(* IEC 61131-3 sources: CodigoPPC/FB Controle, 12 files *)

(* ---- FB_Controle.st ---- *)
(*
   FB_Controle: Bloco Principal de Controle de Exportação (Zero Grid / Limitação).

   OBJETIVO:
   Gerenciar a potência ativa e reativa dos inversores para garantir que a exportação
   de energia no ponto de conexão (PCC) não ultrapasse os limites definidos na agenda.

   ESTRATÉGIA DE CONTROLE (Lógica Inversa):
   - PV (Process Variable) é o valor medido no ponto de conexão
     - Valor Positivo (+) = Importando da rede (Consumo > Geração).
     - Valor Negativo (-) = Exportando para rede (Geração > Consumo).
   - SP (Set Point) é o limite de exportação (ex: -50kW).
   - O PID atua para manter PV >= SP.
     - Se PV > SP (Importando), o PID aumenta a geração.
     - Se PV < SP (Exportando), o PID reduz a geração.
	 Controle de Exportação em kW (Zero = Autoconsumo, Negativo = Exportação, Positivo = Importação).
	Erro: SP - PV.
	Ex: Quero exportar -10kW. Medidor lê +5kW (Importando). Erro = -10 - 5 = -15.
	Para aumentar a geração (reduzir a importação), o PID precisa agir.
	Atenção: Como o comando do inversor é sempre positivo (0..100% de geração), a lógica interna do PI deve ser Inversa (Erro negativo -> Aumenta Saída) ou ajustamos o sinal do erro na entrada.

	No código abaixo, a estratégia usada foi de Normalizar o Erro para "Quanto falta gerar".
	Se o medidor diz +10kW (Importando), precisamos gerar +10kW a mais.
	Se o medidor diz -20kW (Exportando muito) e o limite é -10kW, precisamos gerar 10kW a menos.

    Hierarquia de prioridades ou objetivos:

    Prioridade 1: MAXIMIZAR P (Potência Ativa)
	Objetivo: Gerar o máximo de potência ativa possível
	Limite: Exportação máxima (agenda + safety margin + limite de fase)
	Flexibilidade: RÍGIDO - nunca exceder

	Prioridade 2: PF ≥ 0.92 NO PONTO DE CONEXÃO
	Objetivo: Manter fator de potência ≥ 0.92 (indutivo)
	Método: Compensar Q da carga com Q dos inversores
	Flexibilidade: SOFT - sinaliza se não conseguir, mas NÃO reduz P

	Prioridade 3: BALANCEAMENTO DE FASES

    Ordem de execução:
	0. Leitura do medidor e ajuste dos valores para unidades corretas
	Lê registradores Modbus, converte e armazena como variáveis Globais

	Dentro de FB_Controle
	1. FB_Scheduler - Define limite de exportação baseado em datas, dias de semana e horário
    2. FB_PowertController
		2.1. PI → P_cmd_raw
    	2.2. Safety Margin → P_cmd_with_margin
    	2.3. Limitador de Fase → P_cmd_limited
    3. FB_FFQ - Feedforward de Q (estimativa inicial)
    4. FB_PIQ - Controlador PI de fator de potência
	5. FB_PAlloc - Aloca P pelos inversores
    6. FB_QAlloc - Aloca Q pelos inversores
	7. FB_Diagnostico
	8. STATUS DE PF
*)
FUNCTION_BLOCK FB_Controle
VAR_INPUT
    bReset : BOOL;
END_VAR

VAR
    // ════════════════════════════════════════════════════════════
    // SUBSISTEMAS (Function Blocks)
    // ════════════════════════════════════════════════════════════
    fbScheduler 			: FB_Scheduler;
    fbPowerCtrl 			: FB_PowerController;   // ✅ NOVO: Substitui fbPI + fbSafetyMargin + fbFLimiter
    fbFFQ 					: FB_FFQ;
    fbPIQ 					: FB_PIQ;
    fbPAlloc 				: FB_PAlloc;
    fbQAlloc 				: FB_QAlloc;
    fbDiagnostico 			: FB_Diagnostico;

    // ════════════════════════════════════════════════════════════
    // VARIÁVEIS DE TRABALHO
    // ════════════════════════════════════════════════════════════
    PF_measured 			: REAL;
    Q_cmd_kvar 				: REAL;
    Q_feedforward_kvar 		: REAL;
    bQ_limit_reached 		: BOOL := FALSE;
    bP_limit_reached 		: BOOL := FALSE;
	rPcmd_kW				: REAL;
	rPallocSum_kW			: REAL;
END_VAR

    // ════════════════════════════════════════════════════════════════
    // 0. VERIFICAÇÕES INICIAIS E INICIALIZAÇÃO
    // ════════════════════════════════════════════════════════════════

    // Fator de potência medido (valor absoluto)
    PF_measured := ABS(GVL_Main.PFt);

    // ════════════════════════════════════════════════════════════════
    // 1. FB_SCHEDULER - Define Limite de Exportação
    // ════════════════════════════════════════════════════════════════

    IF GVL_Pers.OperationMode THEN
    	GVL_Main.MaxExportLimit:=0;				// TRUE = Zero Grid (exportação zero)
    ELSE
    	fbScheduler();   						// Global.MaxExportLimit definido a partir das agendas de horarios no Scheduller
    END_IF

    // ────────────────────────────────────────────────────────────────
    // 2. CONTROLADOR DE POTÊNCIA ATIVA (PI + Safety + Limites)
    // ────────────────────────────────────────────────────────────────

    fbPowerCtrl(
        ExportLimit_kW := GVL_Main.MaxExportLimit,
        Feedback_kW := GVL_Main.Pt,
        bReset := bReset
    );

    bP_limit_reached := fbPowerCtrl.bPhase_limited OR fbPowerCtrl.bSaturated;
    // ════════════════════════════════════════════════════════════════
    // 3. FB_FFQ - Feedforward de Q
    // ════════════════════════════════════════════════════════════════

    // Calcula Q necessário para manter PF = 0.92 com a potência comandada
    fbFFQ(
        P_active_kW := fbPowerCtrl.P_cmd_kW,
        PF_target_abs := GVL_Pers.PF_target,
        PF_sign := -1.0                              // capacitivo (negativo)
    );

    Q_feedforward_kvar := fbFFQ.Q_reactive_kvar;

    // ════════════════════════════════════════════════════════════════
    // 4. FB_PIQ - Controle de Fator de Potência
    // ════════════════════════════════════════════════════════════════

    // Controlador PI de fator de potência
    fbPIQ(
        SP := GVL_Pers.PF_target,         							// Setpoint de PF (0.92)
        PV := PF_measured,              							// PF medido (absoluto)
    	Kp:= GVL_Pers.Kp_Q,
    	Ki:= GVL_Pers.Ki_Q,
    	CycleTime:= GVL_Main.ControlCycle,
        P_cmd := fbPowerCtrl.P_cmd_kW,     							// Comando de P (para referência)
        RampUp := GVL_Pers.RampUp_Q,      							// Rampa de subida (kvar/s)
        RampDown := GVL_Pers.RampDown_Q,  							// Rampa de descida (kvar/s)
        DeadbandAbs := GVL_Pers.Deadband_Q, 							// Zona morta de PF
        Reset := bReset,                 							// Reset
    	bExternal_Saturated := bQ_limit_reached OR bP_limit_reached // FEEDBACK do ciclo anterior - calculado em fbQAlloc.
    );

    Q_cmd_kvar := Q_feedforward_kvar + fbPIQ.MV;  // Comando de Q em kvar

    // Clamp superior: não pode exceder Q máximo dos inversores
    IF Q_cmd_kvar > GVL_Main.Q_max_permitido THEN
        Q_cmd_kvar := GVL_Main.Q_max_permitido;
    END_IF
    // Clamp inferior: se PF_sign = indutivo, Q não pode ser negativo
    IF Q_cmd_kvar < 0.0 THEN
        Q_cmd_kvar := 0.0;  // Não permite Q negativo (capacitivo) se não desejado
    END_IF

    // ════════════════════════════════════════════════════════════════
    // 5. FB_PAlloc - Aloca P (PRIORIDADE MÁXIMA)
    // ══════════���═════════════════════════════════════════════════════

    fbPAlloc(
        P_total_cmd_kW := fbPowerCtrl.P_cmd_kW
    );
    // WARN_P_ALLOC_SATURATED = P alocado < P comandado
    rPcmd_kW:= ABS(fbPowerCtrl.P_cmd_kW);
    rPallocSum_kW:= ABS(fbPowerCtrl.P_cmd_kW);
    IF rPcmd_kW < rPallocSum_kW THEN
    	FC_LogEvent(eCode:=E_EventCode.WARN_P_ALLOC_SATURATED,bRaised:=TRUE,rParam1:=rPcmd_kW,rParam2:=rPallocSum_kW,uMachState := GVL_Main.MachineState);
    END_IF
    GVL_Main.P_allocated_kW := fbPAlloc.P_allocated_kW;

    // ════════════════════════════════════════════════════════════════
    // 6. FB_QAlloc - Aloca Q
    // ════════════════════════════════════════════════════════════════

    fbQAlloc(
        Q_total_cmd_kvar := Q_cmd_kvar
    );

    GVL_Main.Q_allocated_kvar := fbQAlloc.Q_allocated_kvar;

    // Armazena flag de saturação para próximo ciclo
    bQ_limit_reached := fbQAlloc.bQ_limit_reached;

    GVL_Alarm.ALARM_Q_LIMITED_BY_SMAX := bQ_limit_reached;
    IF GVL_Alarm.ALARM_Q_LIMITED_BY_SMAX THEN
    	FC_LogEvent(eCode:=E_EventCode.WARN_Q_LIMITED_BY_SMAX,bRaised:=TRUE,rParam1:=Q_cmd_kvar,rParam2:=fbQAlloc.Q_allocated_kvar,uMachState := GVL_Main.MachineState);
    END_IF

    // ════════════════════════════════════════════════════════════════
    // 7. FB_Diagnostico - Gera diagnóstico completo
    // ════════════════════════════════════════════════════════════════

    fbDiagnostico(
        P_allocated_kW := fbPAlloc.P_allocated_kW,
        Q_commanded_kvar := Q_cmd_kvar,
        Q_allocated_kvar := fbQAlloc.Q_allocated_kvar,
        Q_capacity_kvar := fbQAlloc.Q_capacity_total,
        PF_measured := PF_measured,
        PF_achieved := fbQAlloc.PF_effective,
        bQ_limited := fbQAlloc.bQ_limit_reached
    );

    // ────────────────────────────────────────────────────────────────
    // 8. STATUS DE PF
    // ────────────────────────────────────────────────────────────────
    GVL_Alarm.ALARM_PF_BELOW_TARGET:= (fbQAlloc.PF_effective < GVL_Pers.PF_target);
    IF GVL_Alarm.ALARM_PF_BELOW_TARGET THEN
    	FC_LogEvent(
    		eCode:=E_EventCode.WARN_PF_BELOW_TARGET,
    		bRaised:=TRUE,
    		rParam1:=fbQAlloc.PF_effective,
    		rParam2:=GVL_Pers.PF_target,
    		uMachState := GVL_Main.MachineState
    		);
    END_IF

END_FUNCTION_BLOCK

(* ---- FB_Diagnostico.st ---- *)
(*
    ════════════════════════════════════════════════════════════════
    FB_Diagnostico - Diagnóstico de Fator de Potência
    ════════════════════════════════════════════════════════════════

    Gera diagnóstico completo do sistema de compensação de PF,
    incluindo alarmes, recomendações e estatísticas.

    ═══���════════════════════════════════════════════════════════════
*)

FUNCTION_BLOCK FB_Diagnostico
VAR_INPUT
    P_allocated_kW : REAL;
    Q_commanded_kvar : REAL;
    Q_allocated_kvar : REAL;
    Q_capacity_kvar : REAL;
    PF_measured : REAL;
    PF_achieved : REAL;
    bQ_limited : BOOL;
END_VAR

VAR
    Q_deficit : REAL;
    Q_deficit_pct : REAL;
    S_total_avail : REAL;
    S_total_used : REAL;
    bank_size : REAL;
    bank_size_int : DINT;  // ✅ DINT (não INT)
END_VAR

    // ════════════════════════════════════════════════════════════════
    // 1. ARMAZENA VALORES BÁSICOS
    // ════════════════════════════════════════════════════════════════

    GVL_Main.P_generated_kW := P_allocated_kW;
    GVL_Main.P_allocated_kW := P_allocated_kW;
    GVL_Main.Q_commanded_kvar := Q_commanded_kvar;
    GVL_Main.Q_allocated_kvar := Q_allocated_kvar;
    GVL_Main.Q_available_kvar := Q_capacity_kvar;
    GVL_Main.PF_measured := PF_measured;
    GVL_Main.PF_achieved := PF_achieved;

    // Q medido (do ponto de conexão)
    GVL_Main.Q_measured_kvar := GVL_Main.Qt;  // Já convertido em kvar pelo FB_AjustaLeitura

    // ════════════════════════════════════════════════════════════════
    // 2. CALCULA DÉFICIT DE Q
    // ════════════════════════════════════════════════════════════════

    Q_deficit := Q_commanded_kvar - Q_allocated_kvar;
    GVL_Main.Q_deficit_kvar := Q_deficit;

    // Déficit percentual
    IF ABS(Q_commanded_kvar) > 0.1 THEN
        Q_deficit_pct := (ABS(Q_deficit) / ABS(Q_commanded_kvar)) * 100.0;
    ELSE
        Q_deficit_pct := 0.0;
    END_IF
    GVL_Main.Q_deficit_percent := Q_deficit_pct;

    // ════════════════════════════════════════════════════════════════
    // 3. CALCULA UTILIZAÇÃO DE S
    // ════════════════════════════════════════════════════════════════

    // S total disponível
    S_total_avail := GVL_Main.InstalledSmax;
    GVL_Main.S_total_available_kVA := S_total_avail;

    // S total usado
    S_total_used := SQRT((P_allocated_kW * P_allocated_kW) + (Q_allocated_kvar * Q_allocated_kvar));
    GVL_Main.S_total_used_kVA := S_total_used;

    // Utilização percentual
    IF S_total_avail > 0.0 THEN
        GVL_Main.S_utilization_pct := (S_total_used / S_total_avail) * 100.0;
    ELSE
        GVL_Main.S_utilization_pct := 0.0;
    END_IF

    // ════════════════════════════════════════════════════════════════
    // 4. CALCULA UTILIZAÇÃO DE Q
    // ════════════════════════════════════════════════════════════════

    GVL_Main.Q_capacity_total_kvar := Q_capacity_kvar;

    IF Q_capacity_kvar > 0.0 THEN
        GVL_Main.Q_utilization_pct := (ABS(Q_allocated_kvar) / Q_capacity_kvar) * 100.0;
    ELSE
        GVL_Main.Q_utilization_pct := 0.0;
    END_IF

    // ════════════════════════════════════════════════════════════════
    // 5. CALCULA TAMANHO DE BANCO DE CAPACITORES
    // ════════════════════════════════════════════════════════════════

    IF Q_deficit > 0.1 THEN
        // Adiciona 10% de margem
        bank_size := ABS(Q_deficit) * 1.1;
    	bank_size := DINT_TO_REAL(TRUNC(bank_size / 5.0) + 1) * 5.0;
        GVL_Main.Capacitor_bank_size_kvar := bank_size;
        GVL_Main.Capacitor_bank_recommended := TRUE;
    ELSE
        GVL_Main.Capacitor_bank_size_kvar := 0.0;
        GVL_Main.Capacitor_bank_recommended := FALSE;
    END_IF

    // ════════════════════════════════════════════════════════════════
    // 6. DETERMINA STATUS DE PF
    // ════════════════════════════════════════════════════════════════

    IF PF_achieved >= GVL_Main.PF_target THEN
        GVL_Main.PF_OK := TRUE;
        GVL_Main.PFErro := FALSE;
        GVL_Main.PF_alarm_code := 0;  // OK
    ELSE
        GVL_Main.PF_OK := FALSE;

        IF bQ_limited THEN
            GVL_Main.PFErro := TRUE;

            // Classifica severidade
            IF Q_deficit_pct > 20.0 THEN
                GVL_Main.PF_alarm_code := 2;  // Crítico
    			FC_LogEvent(
    				eCode:=E_EventCode.ALARM_Q_LIMITED_SURPASS,
    				bRaised:=TRUE,
    				rParam1:=0.0,
    				rParam2:=0.0,
    				uMachState := GVL_Main.MachineState
    				);
            ELSE
                GVL_Main.PF_alarm_code := 1;  // Aviso
    			FC_LogEvent(
    				eCode:=E_EventCode.ALARM_Q_LIMITED_REACHED,
    				bRaised:=TRUE,
    				rParam1:=0.0,
    				rParam2:=0.0,
    				uMachState := GVL_Main.MachineState
    				);
            END_IF
        ELSE
            // PF < 0.92 mas não por limite de Q (transitório)
            GVL_Main.PFErro := FALSE;
            GVL_Main.PF_alarm_code := 1;
        END_IF
    END_IF

    // ════════════════════════════════════════════════════════════════
    // 7. ATUALIZA HISTÓRICO (OPCIONAL - implementar com timers)
    // ════════════════════════════════════════════════════════════════

    // Atualiza PF mínimo
    IF PF_achieved < GVL_Main.PF_min_24h THEN
        GVL_Main.PF_min_24h := PF_achieved;
    END_IF

    // Atualiza déficit máximo
    IF Q_deficit > GVL_Main.Q_deficit_max_24h THEN
        GVL_Main.Q_deficit_max_24h := Q_deficit;
    END_IF

    // Conta alarmes (incrementar quando alarme dispara pela primeira vez)
    // (Implementar com edge detection)
END_FUNCTION_BLOCK

(* ---- FB_DroopP.st ---- *)
(*
    FB_DroopP - Droop para Potência Ativa
    Gera um comando base proporcional ao erro de potência.
    Uso: antes do PI (PI corrige residual).
*)
FUNCTION_BLOCK FB_DroopP
VAR_INPUT
    Enable        : BOOL;   // Habilita droop
    bReset        : BOOL;   // Reset do droop
    Error_kW      : REAL;   // Erro (Setpoint - Feedback)
    K_droop       : REAL;   // Ganho droop (kW/kW)
    Deadband_kW   : REAL;   // Zona morta
    P_max_kW      : REAL;   // Limite absoluto do droop (kW)
END_VAR

VAR_OUTPUT
    P_droop_kW    : REAL;   // Saída do droop (kW)
END_VAR

VAR
    P_cmd : REAL;
    erro  : REAL;
END_VAR

    // ──────────────────────────────────��───────────────────────────
    // Reset
    // ──────────────────────────────────────────────────────────────
    IF bReset THEN
        P_droop_kW := 0.0;
        RETURN;
    END_IF

    // ──────────────────────────────────────────────────────────────
    // Lógica do droop
    // ──────────────────────────────────────────────────────────────
    IF NOT Enable THEN
        P_droop_kW := 0.0;
        RETURN;
    END_IF

    // Aplica deadband ao erro
    erro := Error_kW;
    IF ABS(erro) < Deadband_kW THEN
        erro := 0.0;
    END_IF

    P_cmd := K_droop * erro;

    // Limite absoluto
    IF P_cmd > P_max_kW THEN
        P_cmd := P_max_kW;
    ELSIF P_cmd < -P_max_kW THEN
        P_cmd := -P_max_kW;
    END_IF

    P_droop_kW := P_cmd;
END_FUNCTION_BLOCK

(* ---- FB_FFQ.st ---- *)
(*
    FB_FFQ - Feedforward de Potência Reativa

    Calcula o Q MÍNIMO necessário para que a SAÍDA DOS INVERSORES
    atinja PF_target quando gerando P_active_kW.

    IMPORTANTE:
    - NÃO usa medição do PCC (isso é responsabilidade do FB_PIQ)
    - Fornece estimativa inicial (feedforward)
    - PIQ corrige com base no PF medido (feedback)

    ════════════════════════════════════════════════════════════════
    LÓGICA CORRETA (GD Solar com Carga Indutiva):
    ════════════════════════════════════════════════════════════════

    1. Medidor no PCC lê:
       - P_medido (importação/exportação)
       - Q_medido (da carga, tipicamente INDUTIVO +)

    2. Para atingir PF = 0.92 no PCC:
       Q_permitido = |P_medido| × tan(acos(0.92))
                   = |P_medido| × 0.4256

    3. Inversores devem compensar Q da carga:
       Q_inv = Q_medido - Q_permitido

    EXEMPLO:
    ────────────────────────────────────────────────────────────────
    P_medido = -100 kW (exportando)
    Q_medido = +300 kvar (carga indutiva)

    Q_permitido = 100 × 0.4256 = 42.56 kvar
    Q_inv = 300 - 42.56 = 257.44 kvar CAPACITIVO

    → Inversores fornecem -257.44 kvar (CAPACITIVO)
    → PF_pcc = 100 / √(100² + 42.56²) ≈ 0.92 ✅
    ════════════════════════════════════════════════════════════════

*)

FUNCTION_BLOCK FB_FFQ
VAR_INPUT
    P_active_kW   : REAL;    // Potência ativa comandada (kW)
    PF_target_abs : REAL;    // PF alvo (0.92)
    PF_sign       : REAL;    // 1.0 = indutivo, -1.0 = capacitivo
END_VAR

VAR_OUTPUT
    Q_reactive_kvar : REAL;   // Potência Reativa Calculada (var) - Q mínimo para atingir PF_target
END_VAR

VAR
    tan_phi : REAL;           // Tangente do ângulo de fase
    Q_target    : REAL;       // Q total necessário no ponto de conexão
END_VAR

    // Proteção: se potência ativa é zero ou negativa, não há Q a calcular
    IF P_active_kW <= 0.0 THEN
        Q_reactive_kvar := 0.0;
        RETURN;
    END_IF

    // Proteção: PF_target deve estar entre 0 e 1
    IF PF_target_abs <= 0.0 OR PF_target_abs > 1.0 THEN
        Q_reactive_kvar := 0.0;
        RETURN;
    END_IF

    // Q total necessário no ponto de conexão para PF = 0.92
    // Método 1: usando tan(acos(PF))
    // phi := ACOS(PF_target_abs);              // Ângulo de fase em radianos
    // tan_phi := TAN(phi);                     // Tangente do ângulo
    // Q_reactive_var := P_active_W * tan_phi;
    // Método 2: Simplificado (mais eficiente, evita ACOS e TAN)
    // tan(acos(x)) = sqrt(1 - x²) / x
    tan_phi := SQRT(1.0 - (PF_target_abs * PF_target_abs)) / PF_target_abs;
    Q_target := P_active_kW * tan_phi;

    // atribuição correta
    Q_reactive_kvar := Q_target;

    // Aplica o sinal (Indutivo = positivo, Capacitivo = negativo)
    // - Cargas normalmente são INDUTIVAS (consomem Q+)
    // - Inversores devem fornecer Q CAPACITIVO (Q-) para compensar
    // - PF_sign é configurável para casos especiais (ex: carga capacitiva)
    //
    // REGRA:
    // - PF_sign > 0 → Q positivo (inversor fornece Q indutivo - raro)
    // - PF_sign < 0 → Q negativo (inversor fornece Q capacitivo - normal)
    // Nota: Para controle de exportação, normalmente usamos capacitivo (negativo)

        IF PF_sign < 0.0 THEN
            Q_reactive_kvar := -Q_target;  // Capacitivo
        ELSE
            Q_reactive_kvar := Q_target;   // Indutivo
        END_IF

    // Resultado: Q_reactive_var é o Q MÍNIMO para atingir PF_target
    // - Se injetar menos Q: PF > PF_target (melhor)
    // - Se injetar mais Q: PF < PF_target (pior)
    // - Se injetar exatamente Q: PF = PF_target
END_FUNCTION_BLOCK

(* ---- FB_FLimiter.st ---- *)
(*
    FB_FLimiter - Limitador por Fase

    Função:
    - Verifica se o comando causaria EXPORTAÇÃO excessiva em alguma fase
    - Se fase está IMPORTANDO: ignora (não há problema)
    - Se fase está EXPORTANDO: verifica se comando excederia limite

    Lógica:
    1. Calcula P futuro por fase = P_atual + (P_cmd / 3)
    2. Para cada fase EXPORTANDO (P < 0):
       - Verifica se P_futuro < P_phase_limit (mais exportação que permitido)
       - Se sim, calcula comando máximo para essa fase
    3. Usa o MENOR comando máximo entre as fases

    Convenção de sinais:
    - P > 0: Importação
    - P < 0: Exportação
    - MaxExportLimit: VALOR POSITIVO na agenda (ex: 90 kW)
    - P_phase_limit: NEGATIVO internamente (ex: -30 kW)

    Exemplo:
    - Agenda: MaxExportLimit = 90 kW (sem sinal)
    - Internamente: P_phase_limit = -90/3 = -30 kW por fase
    - Se Pa = -25 kW (exportando 25 kW)
    - Se P_cmd = -18 kW (quer aumentar exportação)
    - P_future_A = -25 + (-18/3) = -31 kW → EXCEDE -30 kW → LIMITA
*)

FUNCTION_BLOCK FB_FLimiter
VAR_INPUT
    P_cmd_in : REAL;                // Comando de P calculado pelo PI (kW)
    PowerMode : UINT;               // 0=Total, 1=Por fase, 2=Ambos
END_VAR

VAR_OUTPUT
    P_cmd_out : REAL;               // Comando de P limitado por fase (kW)
    bPhase_limited : BOOL;          // TRUE = alguma fase limitou
	sLimited_phase : STRING;        // Qual fase limitou: 'A', 'B', 'C', 'AB', etc.
END_VAR

VAR
    P_cmd_per_phase : REAL;         // Comando adicional por fase (kW)
    P_future_A : REAL;              // P futuro na fase A após aplicar comando (kW)
    P_future_B : REAL;              // P futuro na fase B após aplicar comando (kW)
    P_future_C : REAL;              // P futuro na fase C após aplicar comando (kW)
    P_phase_limit : REAL;           // Limite de exportação por fase (kW negativo)
    P_max_cmd_A : REAL;             // Comando máximo permitido para fase A (kW)
    P_max_cmd_B : REAL;             // Comando máximo permitido para fase B (kW)
    P_max_cmd_C : REAL;             // Comando máximo permitido para fase C (kW)
    P_max_cmd_total : REAL;         // Comando máximo total permitido (kW)
	NO_LIMIT : REAL;                // Constante para "sem limite"
    bLimitA : BOOL;                 // Fase A está limitando
    bLimitB : BOOL;                 // Fase B está limitando
    bLimitC : BOOL;                 // Fase C está limitando
END_VAR

    // Comando adicional por fase (distribuído equilibradamente)
    P_cmd_per_phase := P_cmd_in / 3.0;

    // Limite de exportação por fase
    // Se MaxExportLimit = -90 kW, então por fase = -30 kW
    P_phase_limit := -ABS(GVL_Main.MaxExportLimit) / 3.0;

    // ════════════════════════════════════════════════════════════════
    // ════════════════════════════════════════════════════════════════
    // Inicialização
    // ════════════════════════════════════════════════════════════════
    NO_LIMIT := GVL_Main.InstalledPower * 10.0;  // Valor grande, mas realista
    sLimited_phase := '';
    bLimitA := FALSE;
    bLimitB := FALSE;
    bLimitC := FALSE;

    // ════════════════════════════════════════════════════════════════
    // Se PowerMode = 0, não verifica fase
    // ════════════════════════════════════════════════════════════════
    IF PowerMode = 0 THEN
        P_cmd_out := P_cmd_in;
        bPhase_limited := FALSE;
        RETURN;
    END_IF

    // ════════════════════════════════════════════════════════════════
    // Proteção: Se InstalledPower não configurado
    // ════════════════════════════════════════════════════════════════
    IF GVL_Main.InstalledPower <= 0.0 THEN
        P_cmd_out := 0.0;
        bPhase_limited := TRUE;
        sLimited_phase := 'ERROR: InstalledPower=0';
        RETURN;
    END_IF

    // ════════════════════════════════════════════════════════════════
    // Calcula P futuro em cada fase após aplicar comando
    // ════════════════════════════════════════════════════════════════
    P_future_A := GVL_Main.Pa + P_cmd_per_phase;
    P_future_B := GVL_Main.Pb + P_cmd_per_phase;
    P_future_C := GVL_Main.Pc + P_cmd_per_phase;

    // ════════════════════════════════════════════════════════════════
    // Verifica FASE A
    // ════════════════════════════════════════════════════════════════
    IF P_future_A < 0.0 THEN
        // Fase A estará EXPORTANDO após aplicar comando

        IF P_future_A < P_phase_limit THEN
            // Excederia o limite de exportação!
            // Calcula quanto PODE aumentar exportação sem exceder:
            // P_max_per_phase = P_limit - P_atual
            // P_max_total = P_max_per_phase * 3
            P_max_cmd_A := (P_phase_limit - GVL_Main.Pa) * 3.0;
            bLimitA := TRUE;
        ELSE
            // Dentro do limite: sem restrição
            P_max_cmd_A := NO_LIMIT;
        END_IF

    ELSE
        // Fase A estará IMPORTANDO: sem problema
        P_max_cmd_A := NO_LIMIT;
    END_IF

    // ════════════════════════════════════════════════════════════════
    // Verifica FASE B
    // ════════════════════════════════════════════════════════════════
    IF P_future_B < 0.0 THEN
        // Fase B estará EXPORTANDO

        IF P_future_B < P_phase_limit THEN
            P_max_cmd_B := (P_phase_limit - GVL_Main.Pb) * 3.0;
            bLimitB := TRUE;
        ELSE
            P_max_cmd_B := NO_LIMIT;
        END_IF

    ELSE
        // Fase B estará IMPORTANDO
        P_max_cmd_B := NO_LIMIT;
    END_IF

    // ════════════════════════════════════════════════════════════════
    // Verifica FASE C
    // ════════════════════════════════════════════════════════════════
    IF P_future_C < 0.0 THEN
        // Fase C estará EXPORTANDO

        IF P_future_C < P_phase_limit THEN
            P_max_cmd_C := (P_phase_limit - GVL_Main.Pc) * 3.0;
            bLimitC := TRUE;
        ELSE
            P_max_cmd_C := NO_LIMIT;
        END_IF

    ELSE
        // Fase C estará IMPORTANDO
        P_max_cmd_C := NO_LIMIT;
    END_IF

    // ════════════════════════════════════════════════════════════════
    // Aplica o MENOR limite (fase mais restritiva)
    // ════════════════════════════════════════════════════════════════
    P_max_cmd_total := MIN(P_max_cmd_A, MIN(P_max_cmd_B, P_max_cmd_C));

    // ════════════════════════════════════════════════════════════════
    // Verifica se houve limitação
    // ════════════════════════════════════════════════════════════════
    IF P_cmd_in > P_max_cmd_total THEN
        P_cmd_out := P_max_cmd_total;
        bPhase_limited := TRUE;

        // Identifica qual(is) fase(s) limitou
        IF bLimitA THEN sLimited_phase := CONCAT(sLimited_phase, 'A'); END_IF
        IF bLimitB THEN sLimited_phase := CONCAT(sLimited_phase, 'B'); END_IF
        IF bLimitC THEN sLimited_phase := CONCAT(sLimited_phase, 'C'); END_IF

    ELSE
        P_cmd_out := P_cmd_in;
        bPhase_limited := FALSE;
        sLimited_phase := '';
    END_IF
END_FUNCTION_BLOCK

(* ---- FB_PAlloc.st ---- *)
(*
    ════════════════════════════════════════════════════════════════
    FB_PAlloc - Alocador de Potência Ativa (PRIORIDADE MÁXIMA)
    ════════════════════════════════════════════════════════════════
*)
FUNCTION_BLOCK FB_PAlloc
VAR_INPUT
    P_total_cmd_kW : REAL;          // Comando de P total (do FB_PI)
END_VAR

VAR_OUTPUT
    P_allocated_kW : REAL;          // ✅ ADICIONAR ESTA SAÍDA!
END_VAR

VAR
    i : UINT;
    P_target_i : REAL;
    P_actual_i : REAL;
    P_total_calc : REAL;
    proportion : REAL;
END_VAR

    P_total_calc := 0.0;

    FOR i := 1 TO GVL_Main.NMAXINVERSORES DO

        IF GVL_Pers.InvActivePower[i] > 0.0 THEN

            // Proporção do inversor
            proportion := GVL_Pers.InvActivePower[i] / GVL_Main.InstalledPower;

            // P proporcional
            P_target_i := P_total_cmd_kW * proportion;

            // Limita apenas pela nominal (ignora S_max por enquanto)
            P_actual_i := MIN(P_target_i, GVL_Pers.InvActivePower[i]);

            // Armazena P
            GVL_Main.P_inv_kW[i] := P_actual_i;

            // Setpoint percentual
            IF GVL_Pers.InvActivePower[i] > 0.0 THEN
                GVL_Main.P_inv_Percent[i] := (P_actual_i / GVL_Pers.InvActivePower[i]) * 100.0;
            ELSE
                GVL_Main.P_inv_Percent[i] := 0.0;
            END_IF

            P_total_calc := P_total_calc + P_actual_i;

        ELSE
            GVL_Main.P_inv_kW[i] := 0.0;
            GVL_Main.P_inv_Percent[i] := 0.0;
        END_IF

    END_FOR

    // ✅ ATUALIZA SAÍDA
    P_allocated_kW := P_total_calc;
END_FUNCTION_BLOCK

(* ---- FB_PI.st ---- *)
FUNCTION_BLOCK FB_PI
VAR_INPUT
    setpoint    : REAL;         		// Setpoint desejado
    feedback    : REAL;         		// Medição atual (feedback)
    Kp          : REAL;         		// Ganho proporcional
    Ki          : REAL;         		// Ganho integral
    OutMax      : REAL;         		// Limite superior de saída
    OutMin      : REAL;         		// Limite inferior de saída
    CycleTime   : REAL;         		// Tempo de ciclo (s)
    RampUp      : REAL := 1.0E+6;  		//  Rampa de subida (unidade/s). Default = sem limite
    RampDown    : REAL := 1.0E+6;  		//  Rampa de descida (unidade/s). Default = sem limite
    Deadband    : REAL := 0.0;          //  deadband em kW (já convertido de %)
    bReset      : BOOL := FALSE;        //  reset do PI
END_VAR

VAR_OUTPUT
    u           : REAL;         		// Saída do controlador
    erro        : REAL;         		// Erro atual (setpoint - feedback)
    bSaturated  : BOOL;         		// TRUE = saída saturada
END_VAR

VAR
    integ           : REAL := 0.0;      // Integral acumulada
    LastOut         : REAL := 0.0;
    erroAtual       : REAL;             // Erro no ciclo atual
    u_prop          : REAL;             // Componente proporcional
    u_raw           : REAL;             // Saída antes da saturação
    u_limited       : REAL;         	// Saída após saturação, antes da rampa
    delta           : REAL;         	// Variação desejada
    delta_max       : REAL;         	// Variação máxima permitida
    primeiro_ciclo  : BOOL := TRUE;     // Flag de primeira execução
    sinal_saturacao : INT;              // +1: saturado max, -1: saturado min, 0: não saturado
END_VAR

    // ════════════════════════════════════════════════════════════════
    // Reset explícito
    // ════════════════════════════════════════════════════════════════
    IF bReset THEN
        integ := 0.0;
        LastOut := 0.0;
        u := 0.0;
        bSaturated := FALSE;
        primeiro_ciclo := TRUE;
        RETURN;
    END_IF

    // ════════════════════════════════════════════════════════════════
    // Inicialização suave na primeira execução
    // ════════════════════════════════════════════════════════════════
    IF primeiro_ciclo THEN
        integ := 0.0;
        primeiro_ciclo := FALSE;

        // Se quiser inicializar LastOut com valor atual do medidor:
        // LastOut := feedback;  // Opcional: evita salto inicial
    END_IF

    // ════════════════════════════════════════════════════════════════
    // Cálculo do Erro + Deadband
    // ════════════════════════════════════════════════════════════════
    erroAtual := setpoint - feedback;

    // ✅ Deadband
    IF ABS(erroAtual) < Deadband THEN
        erroAtual := 0.0;
    END_IF

    erro := erroAtual;  // Saída para diagnóstico

    // ════════════════════════════════════════════════════════════════
    // Componente Proporcional
    // ════════════════════════════════════════════════════════════════
    u_prop := Kp * erroAtual;

    // ════════════════════════════════════════════════════════════════
    // Saída Raw (P + I + LastOut)
    // ══════════════════════════════════════════���═════════════════════
    u_prop := Kp * erroAtual;
    u_raw := u_prop + integ;

    // ════════════════════════════════════════════════════════════════
    // Saturação
    // ════════════════════════════════════════════════════════════════
    IF u_raw > OutMax THEN
        u_limited := OutMax;
        bSaturated := TRUE;
        sinal_saturacao := 1;
    ELSIF u_raw < OutMin THEN
        u_limited := OutMin;
        bSaturated := TRUE;
        sinal_saturacao := -1;
    ELSE
        u_limited := u_raw;
        bSaturated := FALSE;
        sinal_saturacao := 0;
    END_IF

    // ════════════════════════════════════════���═══════════════════════
    // Rate Limiter (Rampa)
    // ════════════════════════════════════════════════════════════════
    delta := u_limited - LastOut;

    IF delta > 0.0 THEN
        delta_max := RampUp * CycleTime;
        IF delta > delta_max THEN
            u := LastOut + delta_max;
        ELSE
            u := u_limited;
        END_IF
    ELSIF delta < 0.0 THEN
        delta_max := RampDown * CycleTime;
        IF ABS(delta) > delta_max THEN
            u := LastOut - delta_max;
        ELSE
            u := u_limited;
        END_IF
    ELSE
        u := u_limited;
    END_IF
    // ════════════════════════════════════════════════════════════════
    // Anti-windup Melhorado (Conditional Integration)
    // ════════════════════════════════════════════════════════════════
    // Regras:
    // 1. NÃO saturado → acumula normALARMente
    // 2. Saturado MAS erro na direção oposta → permite desacumular
    // 3. Saturado E erro na mesma direção → freeze (não acumula)

    IF NOT bSaturated THEN
        // Caso 1: Normal - acumula integral
        integ := integ + (Ki * erroAtual * CycleTime);

    ELSIF (sinal_saturacao = 1 AND erroAtual < 0.0) OR (sinal_saturacao = -1 AND erroAtual > 0.0) THEN
        // Caso 2: Saturado MAS erro está tentando sair da saturação
        // Permite acumular para ajudar a desaturar
        integ := integ + (Ki * erroAtual * CycleTime);

    ELSE
        // Caso 3: Saturado E erro empurrando mais para saturação
        // NÃO acumula (freeze integral)
        // integ permanece inalterado
    END_IF

    // ════════════════════════════════════════════════════════════════
    // Atualiza LastOut
    // ════════════════════════════════════════════════════════════════
    LastOut := u;
END_FUNCTION_BLOCK

(* ---- FB_PIQ.st ---- *)
(*
    FB_PIQ - Controlador PI para Fator de Potência
    Lógica para PF ≥ 0.92:
    - Se PV (PF medido) ≥ SP (PF target): erro = 0 (objetivo atingido)
    - Se PV < SP: erro = SP - PV (precisa aumentar Q)
    Diferente de um PI normal:
    - Erro ZERO quando PF ≥ target (não tenta melhorar além do necessário)
    - Saída é comando de Q (kvar)
*)

FUNCTION_BLOCK FB_PIQ
VAR_INPUT
    SP : REAL;                      		// Setpoint de PF (0.92)
    PV : REAL;                      		// PF medido (absoluto)
	Kp : REAL;
    Ki : REAL;
    CycleTime : REAL;
    P_cmd : REAL;                   		// Comando de P (para referência)
    RampUp : REAL;                  		// Rampa de subida (kvar/s)
    RampDown : REAL;                		// Rampa de descida (kvar/s)
    DeadbandAbs : REAL;             		// Zona morta de PF (ex: 0.01)
    Reset : BOOL;                   		// Zera o controlador
    bExternal_Saturated : BOOL := FALSE;  	// NOVO: Saturação externa (de FB_QAlloc)
	OutMax : REAL := 1000.0;    			// Limite superior de MV (kvar)
    OutMin : REAL := 0.0;       			// Limite inferior de MV (kvar)
END_VAR

VAR_OUTPUT
    MV : REAL;                      // Comando de Q (kvar)
    Error : REAL;                   // BOOL → REAL (valor do erro)
    Saturated : BOOL;               // TRUE = saída saturada
END_VAR

VAR
    integral : REAL := 0.0;         // Acumulador integral
    P_term : REAL;                  // Termo proporcional
    I_term : REAL;                  // Termo integral
    MV_raw : REAL;                  // Saída bruta (antes de rampa)
    MV_prev : REAL := 0.0;          // Saída do ciclo anterior
    delta : REAL;                   // Variação desejada
    delta_max : REAL;               // Variação máxima permitida
    erro : REAL;                    // Erro de PF
    sinal_saturacao : INT;      	// para anti-windup direcional
END_VAR

    // ════════════════════════════════════════════════════════════════
    // 1. RESET
    // ════════════════════════════════════════════════════════════════
    IF Reset THEN
        integral := 0.0;
        MV := 0.0;
        MV_prev := 0.0;
        Error := 0.0;
        Saturated := FALSE;
        RETURN;
    END_IF

    // ════════════════════════════════════════════════════════════════
    // 2. CALCULA ERRO COM LÓGICA ESPECIAL (PF ≥ TARGET)
    // ════════════════════════════════════════════════════════════════

    IF PV >= SP THEN
        erro := 0.0;  // PF medido ≥ PF target: objetivo atingido
    ELSE
        erro := SP - PV;  // PF medido < PF target: precisa corrigir
    END_IF

    Error := erro;  // ✅ Saída do erro

    // ════════════════════════════════════════════════════════════════
    // 3. ZONA MORTA (DEADBAND)
    // ════════════════════════════════════════════════════════════════

    IF ABS(erro) < DeadbandAbs THEN
        erro := 0.0;
    END_IF

    // ════════════════════════════════════════════════════════════════
    // 4. CÁLCULO PI
    // ════════════════════════════════════════════════════════════════

    P_term := Kp * erro;
    I_term := integral + (Ki * erro * CycleTime);
    MV_raw := P_term + I_term;

    // ════════════════════════════════════════════════════════════════
    // 5. ✅ SATURAÇÃO COM OutMax/OutMin (ALTERAÇÃO)
    // ════════════════════════════════════════════════════════════════
    IF MV_raw > OutMax THEN
        MV_raw := OutMax;
        sinal_saturacao := 1;
    ELSIF MV_raw < OutMin THEN
        MV_raw := OutMin;
        sinal_saturacao := -1;
    ELSE
        sinal_saturacao := 0;
    END_IF

    // ════════════════════════════════════════════════════════════════
    // 6. ANTI-WINDUP (Conditional Integration)
    // ════════════════════════════════════════════════════════════════

    IF bExternal_Saturated OR (sinal_saturacao <> 0) THEN
        // Saturado: só acumula se erro empurra para FORA da saturação
        IF (sinal_saturacao = 1 AND erro < 0.0) OR
           (sinal_saturacao = -1 AND erro > 0.0) THEN
            integral := I_term;  // Permite desacumular
        END_IF
        // Caso contrário: integral permanece (freeze)
        Saturated := TRUE;
    ELSE
        integral := I_term;
        Saturated := FALSE;
    END_IF

    // ════════════════════════════════════════════════════════════════
    // 7. RATE LIMITER (Rampa)
    // ════════════════════════════════════════════════════════════════

    delta := MV_raw - MV_prev;

    IF delta > 0.0 THEN
        delta_max := RampUp * GVL_Main.ControlCycle;
        IF delta > delta_max THEN
            MV := MV_prev + delta_max;
        ELSE
            MV := MV_raw;
        END_IF

    ELSIF delta < 0.0 THEN
        delta_max := RampDown * GVL_Main.ControlCycle;
        IF ABS(delta) > delta_max THEN
            MV := MV_prev - delta_max;
        ELSE
            MV := MV_raw;
        END_IF

    ELSE
        MV := MV_raw;
    END_IF

    MV_prev := MV;
END_FUNCTION_BLOCK

(* ---- FB_PowerController.st ---- *)
(*
    ════════════════════════════════════════════════════════════════
    FB_PowerController - Controlador de Potência Ativa
    ════════════════════════════════════════════════════════════════

    Responsabilidade:
    - Calcular comando de P (PI + Safety Margin + Limites de Fase)
    - Encapsular toda lógica relacionada a potência ativa

    Pipeline:
    1. PI → P_cmd_raw
    2. Safety Margin → P_cmd_with_margin
    3. Limitador de Fase → P_cmd_limited

    ════════════════════════════════════════════════════════════════
*)
FUNCTION_BLOCK FB_PowerController
VAR_INPUT
    ExportLimit_kW : REAL;      // Do scheduler (kW)
    Feedback_kW : REAL;         // Leitura do medidor (kW)
    bReset : BOOL;              // Reset do PI
END_VAR

VAR_OUTPUT
    P_cmd_kW : REAL;            // Comando final (kW)
    bSaturated : BOOL;          // PI saturado
    bPhase_limited : BOOL;      // Limitado por fase
    sLimited_phase : STRING;    // Qual fase limitou
    Margin_applied_kW : REAL;   // Margem aplicada (telemetria)
	EffectiveExportLimit_kW : REAL;
END_VAR

VAR
    // Sub-blocos
    fbPI : FB_PI;
    fbSafetyMargin : FB_SafetyMargin;
    fbFLimiter : FB_FLimiter;
	fbDroop : FB_DroopP;

    // Variáveis internas
    P_setpoint : REAL;
    P_cmd_raw : REAL;
    P_cmd_with_margin : REAL;
	lastInstalledPower : REAL := -1.0;

	// Droop
    P_error_kW : REAL;
    P_droop_kW : REAL;

    P_droop_max_kW : REAL;
    P_cmd_sum : REAL;

	// ✅ Deadband em kW (convertido de %)
	Deadband_P_kW     : REAL;
    Droop_Deadband_kW : REAL;
END_VAR

    // ────────────────────────────────────────────────────────────────
    // ETAPA 1: CONTROLADOR PI
    // ────────────────────────────────────────────────────────────────

    // Setpoint negativo (exportação)
    P_setpoint := -ABS(ExportLimit_kW);

    // Erro (kW)
    P_error_kW := Feedback_kW - P_setpoint;

    // Converte deadband (%) para kW (mínimo 1 kW)
    // Recalcula apenas se InstalledPower mudou
    IF lastInstalledPower <> GVL_Main.InstalledPower THEN
        Deadband_P_kW := MAX(1.0, GVL_Main.InstalledPower * (GVL_Persis.Deadband_P / 100.0));
        Droop_Deadband_kW := MAX(1.0, GVL_Main.InstalledPower * (GVL_Persis.Deadband_Droop / 100.0));
    	Deadband_P_kW := MIN(20.0, MAX(1.0, GVL_Main.InstalledPower * (GVL_Persis.Deadband_P / 100.0)));
    	Droop_Deadband_kW := MIN(20.0, MAX(1.0, GVL_Main.InstalledPower * (GVL_Persis.Deadband_Droop / 100.0)));
        lastInstalledPower := GVL_Main.InstalledPower;
    END_IF

    // Limite máximo do droop (fração da potência instalada)
    P_droop_max_kW := GVL_Persis.Droop_Max * GVL_Main.InstalledPower;

    // Calcula droop
    fbDroop(
        Enable      := GVL_Persis.Droop_Enable,
        bReset      := bReset,
        Error_kW    := P_error_kW,
        K_droop     := GVL_Persis.K_Droop,
        Deadband_kW := Droop_Deadband_kW,
        P_max_kW    := P_droop_max_kW
    );

    P_droop_kW := fbDroop.P_droop_kW;

    // PI de potência ativa
    fbPI(
        setpoint    := P_error_kW,
        feedback    := 0.0,
        Kp          := GVL_Persis.Kp_P,
        Ki          := GVL_Persis.Ki_P,
        OutMax      := GVL_Main.InstalledPower,
        OutMin      := 0.0,
        CycleTime   := GVL_Main.ControlCycle,
    	RampUp      := GVL_Persis.RampUp_P,
        RampDown    := GVL_Persis.RampDown_P,
        Deadband    := Deadband_P_kW,
    	bReset      := bReset
    );

    // Soma droop + PI
    P_cmd_sum := P_droop_kW + fbPI.u;

    // Comando bruto (segue fluxo normal)
    P_cmd_raw := P_cmd_sum;
    IF P_cmd_raw < 0.0 THEN
        P_cmd_raw := 0.0;
    ELSIF P_cmd_raw > GVL_Main.InstalledPower THEN
        P_cmd_raw := GVL_Main.InstalledPower;
    END_IF
    bSaturated := fbPI.bSaturated;

    // ─────────────────────────────────────────���──────────────────────
    // ETAPA 2: SAFETY MARGIN
    // ────────────────────────────────────────────────────────────────

    fbSafetyMargin(
        P_cmd_raw_kW := P_cmd_raw,
        Margin_pct := GVL_Persis.SafetyMargin_pct,
        TC_Power_kW := GVL_Persis.TC_Power_kW
    );

    P_cmd_with_margin := fbSafetyMargin.P_cmd_adjusted_kW;
    Margin_applied_kW := fbSafetyMargin.Margin_applied_kW;  // ✅ Telemetria
    EffectiveExportLimit_kW := P_setpoint + Margin_applied_kW;
    // ────────────────────────────────────────────────────────────────
    // ETAPA 3: LIMITADOR DE FASE
    // ────────────────────────────────────────────────────────────────

    fbFLimiter(
        P_cmd_in := P_cmd_with_margin,
        PowerMode := GVL_Persis.PowerMode
    );

    P_cmd_kW := fbFLimiter.P_cmd_out;
    bPhase_limited := fbFLimiter.bPhase_limited;
    sLimited_phase := fbFLimiter.sLimited_phase;

    // ────────────────────────────────────────────────────────────────
    // PROTEÇÃO FINAL: Potência Instalada
    // ────────────────────────────────────────────────────────────────

    IF P_cmd_kW > GVL_Main.InstalledPower THEN
        P_cmd_kW := GVL_Main.InstalledPower;
        bSaturated := TRUE;
    END_IF
END_FUNCTION_BLOCK

(* ---- FB_QAlloc.st ---- *)
(*
    ════════════════════════════════════════════════════════════════
    FB_QAlloc - Alocador de Potência Reativa
    ════════════════════════════════════════════════════════════════

   // Protocolo Goodwe:
   //   - Indutivo (Q ≥ 0): Reg 80-100 → PF = Reg/100 (0.80-1.00)
   //   - Capacitivo (Q < 0): Reg 1-20 → PF = (100-Reg)/100 (0.80-0.99)
*)

FUNCTION_BLOCK FB_QAlloc
VAR_INPUT
    Q_total_cmd_kvar : REAL;        // Comando de Q total (do FB_PIQ)
END_VAR

VAR_OUTPUT
    bQ_limit_reached : BOOL;        // TRUE = Não conseguiu alocar todo Q
    Q_allocated_kvar : REAL;        // Q efetivamente alocado
    PF_effective : REAL;            // PF efetivo total resultante
    Q_capacity_total : REAL;        // Capacidade total de Q disponível (kvar)
    S_total_used : REAL;            // S total utilizado (kVA)
END_VAR

VAR

	// ✅ Acumuladores totais
    Q_total : REAL;
    P_total : REAL;
    Q_capacity_total_internal : REAL;
    S_total_used_internal : REAL;

	// ✅ Variáveis por inversor
    Q_target_i : REAL;
    Q_actual_i : REAL;
    Q_max_i : REAL;
    S_available_i : REAL;
    P_actual_i : REAL;

    // ✅ Auxiliares
    i : UINT;
    proportion : REAL;
    S_total : REAL;
    S_i : REAL;  // ✅ S do inversor i (calculado 1 vez)

    PF_abs : REAL;  // PF absoluto (sem sinal)
    PF_reg : REAL;  // Registrador Modbus calculado (1-20 ou 80-100)
END_VAR

    // ════════════════════════════════════════════════════════════════
    // INICIALIZAÇÃO
    // ════════════════════════════════════════════════════════════════

    Q_total := 0.0;
    P_total := 0.0;
    Q_capacity_total_internal := 0.0;
    S_total_used_internal := 0.0;
    bQ_limit_reached := FALSE;

    // ════════════════════════════════════════════════════════════════
    // LOOP PRINCIPAL
    // ════════════════════════════════════════════════════════════════

    FOR i := 1 TO GVL_Main.NMAXINVERSORES DO

        IF GVL_Pers.InvActivePower[i] > 0.0 THEN

            // ────────────────────────────────────────────────────────
            // A. LÊ P JÁ ALOCADO
            // ────────────────────────────────────────────────────────
            P_actual_i := GVL_Main.P_inv_kW[i];

            // ────────────────────────────────────────────────────────
            // B. CALCULA Q MÁXIMO DISPONÍVEL
            // ────────────────────────────────────────────────────────
            S_available_i := GVL_Pers.InvSmaxPower[i];

            IF S_available_i > ABS(P_actual_i) THEN
                Q_max_i := SQRT((S_available_i * S_available_i) - (P_actual_i * P_actual_i));
            ELSE
                Q_max_i := 0.0;
            END_IF

            GVL_Main.Inv_Q_available[i] := Q_max_i;

            // ─────────────────────────────────────────���──────────────
            // C. DISTRIBUI Q PROPORCIONALARMENTE
            // ────────────────────────────────────────────────────────
            IF GVL_Main.P_allocated_kW > 0.01 THEN
                proportion := GVL_Main.P_inv_kW[i] / GVL_Main.P_allocated_kW;
            ELSE
                proportion := 0.0;
            END_IF

            Q_target_i := Q_total_cmd_kvar * proportion;

            // ────────────────────────────────────────────────────────
            // D. LIMITA Q AO DISPONÍVEL
            // ────────────────────────────────────────────────────────
            IF ABS(Q_target_i) > Q_max_i THEN

                IF Q_target_i >= 0.0 THEN
                    Q_actual_i := Q_max_i;
                ELSE
                    Q_actual_i := -Q_max_i;
                END_IF

                bQ_limit_reached := TRUE;
                GVL_Main.Inv_limited[i] := TRUE;

            ELSE
                Q_actual_i := Q_target_i;
                GVL_Main.Inv_limited[i] := FALSE;
            END_IF

            // ────────────────────────────────────────────────────────
            // E. ARMAZENA Q
            // ────────────────────���───────────────────────────────────
            GVL_Main.Q_inv_kvar[i] := Q_actual_i;

            // ────────────────────────────────────────────────────────
            // F. CALCULA S UTILIZADO (✅ UMA VEZ)
            // ────────────────────────────────────────────────────────
            S_i := SQRT((P_actual_i * P_actual_i) + (Q_actual_i * Q_actual_i));

            S_total_used_internal := S_total_used_internal + S_i;

            // Utilização de S (%)
            IF S_available_i > 0.0 THEN
                GVL_Main.Inv_S_utilization[i] := (S_i / S_available_i) * 100.0;
            ELSE
                GVL_Main.Inv_S_utilization[i] := 0.0;
            END_IF

            // ────────────────────────────────────────────────────────
            // G. CALCULA PF INDIVIDUAL
            // ────────────────────────────────────────────────────────
            IF S_i > 0.01 THEN
                GVL_Main.PF_inv[i] := P_actual_i / S_i;
            ELSE
                GVL_Main.PF_inv[i] := 1.0;
            END_IF

            // ────────────────────────────────────────────────────────
            // Protocolo Goodwe:
            //   - Indutivo (Q ≥ 0): Reg 80-100 → PF = Reg/100 (0.80-1.00)
            //   - Capacitivo (Q < 0): Reg 1-20 → PF = (100-Reg)/100 (0.80-0.99)
            // ──────────────────────────────────────────────────────────
            // VALIDAÇÃO DE RANGE FÍSICO
            // ──────────────────────────────────────────────────────────
            PF_abs := ABS(GVL_Main.PF_inv[i]);

            IF PF_abs < 0.80 THEN
            // ❌ CRÍTICO: PF < 0.80 não é suportado pelo inversor
    			IF GVL_Main.Q_inv_kvar[i] >= 0.0 THEN
    				GVL_Main.PF_inv[i] := 0.80;   // Indutivo
    			ELSE
    				GVL_Main.PF_inv[i] := -0.80;  // Capacitivo
    			END_IF
    			FC_LogEvent(
    				eCode := E_EventCode.ALARM_MEAS_PFT_RANGE,  // Reutiliza evento existente
    				bRaised := TRUE,
    				rParam1 := UINT_TO_REAL(i),
    				rParam2 := PF_abs,
    				uMachState := GVL_Main.MachineState
    				);
    			PF_abs := 0.80;

            ELSIF PF_abs > 1.0 THEN
                // ❌ CRÍTICO: PF > 1.0 fisicamente impossível
    			IF GVL_Main.Q_inv_kvar[i] >= 0.0 THEN
    				GVL_Main.PF_inv[i] := 1.0;
    			ELSE
    				GVL_Main.PF_inv[i] := -1.0;
    			END_IF
                FC_LogEvent(
                    eCode := E_EventCode.ALARM_MEAS_PFT_RANGE,
                    bRaised := TRUE,
                    rParam1 := UINT_TO_REAL(i),
                    rParam2 := PF_abs,
                    uMachState := GVL_Main.MachineState
                );
                PF_abs := 1.0;
            END_IF

           // ──────────────────────────────────────────────────────────
           // CONVERSÃO PARA FORMATO MODBUS (Baseado no SINAL de Q)
           // ──────────────────────────────────────────────────────────

           IF GVL_Main.Q_inv_kvar[i] >= 0.0 THEN
                // ── INDUTIVO (Q positivo) → Range 80-100 ──
                PF_reg := PF_abs * 100.0;

                // Clamp no range válido
                IF PF_reg < 80.0 THEN
                    PF_reg := 80.0;
                ELSIF PF_reg > 100.0 THEN
                    PF_reg := 100.0;
           		END_IF

           ELSE
                // ── CAPACITIVO (Q negativo) → Range 1-20 ──
                // Fórmula: Reg = 100 - (PF × 100)
                // Ex: PF 0.90 → Reg = 100 - 90 = 10
                PF_reg := 100.0 - (PF_abs * 100.0);

                // Clamp no range válido
                IF PF_reg < 1.0 THEN
                    PF_reg := 1.0;
                 ELSIF PF_reg > 20.0 THEN
                     PF_reg := 20.0;
                END_IF
           END_IF

           // ──────────────────────────────────────────────────────────
           // ARMAZENA VALOR FINAL
           // ──────────────────────────────────────────────────────────
           GVL_Main.PF_inv_Percent[i] := PF_reg;

    	   // ────────────────────────────────────────────────────────
           // H. ACUMULADORES
           // ────────────────────────────────────────────────────────
           P_total := P_total + P_actual_i;
           Q_total := Q_total + Q_actual_i;
           Q_capacity_total_internal := Q_capacity_total_internal + Q_max_i;

        ELSE
            // Inversor inativo
            GVL_Main.Q_inv_kvar[i] := 0.0;
            GVL_Main.PF_inv[i] := 1.0;
            GVL_Main.Inv_Q_available[i] := 0.0;
            GVL_Main.Inv_S_utilization[i] := 0.0;
            GVL_Main.Inv_limited[i] := FALSE;
            GVL_Main.PF_inv_Percent[i] := 100.0;  // PF = 1.0 em formato Modbus
        END_IF

    END_FOR

    // ════════════════════════════════════════════════════════════════
    // SAÍDAS
    // ════════════════════════════════════════════════════════════════

    Q_allocated_kvar := Q_total;
    Q_capacity_total := Q_capacity_total_internal;
    S_total_used := S_total_used_internal;

    // PF efetivo total
    IF P_total > 0.01 OR ABS(Q_total) > 0.01 THEN
        S_total := SQRT((P_total * P_total) + (Q_total * Q_total));
        PF_effective := P_total / S_total;
    ELSE
        PF_effective := 1.0;
    END_IF
END_FUNCTION_BLOCK

(* ---- FB_SafetyMargin.st ---- *)
(*
    ════════════════════════════════════════════════════════════════
    FB_SafetyMargin - Margem de Segurança para Correção de TC
    ════════════════════════════════════════════════════════════════

    Função:
    - Aplica margem de segurança para compensar erro de TC em baixas correntes
    - Desloca setpoint para lado da importação (garante não exportar)

    Exemplo:
    - P_cmd = 100 kW
    - TC_Power = 329 kW
    - Margin = 3%
    - SafetyMargin = 3% × 329 = 9.87 kW
    - P_adjusted = 100 - 9.87 = 90.13 kW
    ════════════════════════════════════════════════════════════════
*)
FUNCTION_BLOCK FB_SafetyMargin
VAR_INPUT
    P_cmd_raw_kW : REAL;        // Comando sem margem
    Margin_pct : REAL;          // Percentual (ex: 3.0)
    TC_Power_kW : REAL;         // Potência do TC
END_VAR

VAR_OUTPUT
    P_cmd_adjusted_kW : REAL;   // Comando com margem
    Margin_applied_kW : REAL;   // Margem aplicada (para telemetria)
END_VAR

VAR
    SafetyMargin_kW : REAL;
END_VAR

    // ════════════════════════════════════════════════════════════════
    // IMPLEMENTAÇÃO
    // ════════════════════════════════════════════════════════════════
    // 1. Proteção: se TC não configurado, não aplica margem
    IF TC_Power_kW <= 0.0 THEN
        P_cmd_adjusted_kW := P_cmd_raw_kW;
        Margin_applied_kW := 0.0;
        RETURN;
    END_IF

    // 2. Calcula margem em kW
    SafetyMargin_kW := (Margin_pct / 100.0) * TC_Power_kW;

    // 3. Aplica margem (reduz comando)
    P_cmd_adjusted_kW := P_cmd_raw_kW - SafetyMargin_kW;

    // 4. Limita para não ficar negativo
    IF P_cmd_adjusted_kW < 0.0 THEN
        P_cmd_adjusted_kW := 0.0;
    END_IF

    // 5. Armazena margem aplicada (para HMI)
    Margin_applied_kW := SafetyMargin_kW;
END_FUNCTION_BLOCK

(* ---- FB_Scheduler.st ---- *)
(*
    FB_Scheduler
    - Agenda semanal: 24 intervalos por dia, 7 dias.
    - Recebe Hora UTC do sistema e converte internamente para LOCAL (Fuso + DST).
    - Feriados/datas especiais sobrescrevem a agenda.
    - Saída: setpoint % da potência instalada.
*)
FUNCTION_BLOCK FB_Scheduler

VAR
    // ════════════════════════════════════════════════════════════
    // VARIÁVEIS DE TIMESTAMP
    // ════════════════════════════════════════════════════════════
    timestampLocal_UDINT : UDINT;           // ✅ Apenas UDINT (sem DINT)
    offsetSeconds : DINT;                   // Offset em segundos (pode ser negativo)
    offsetSeconds_ABS : UDINT;              // Valor absoluto do offset

    // ════════════════════════════════════════════════════════════
    // CONVERSÕES DE DATA/HORA
    // ════════════════════════════════════════════════════════════
    dtNowLocal : DATE_AND_TIME;
    dataNowLocal : DATE;
    todNowLocal : TOD;
    todAsDword : DWORD;
    hora : INT;
    diadasemana : INT;
	semanaindex : BOOL;

    // ════════════════════════════════════════════════════════════
    // CACHE DE DATAS ESPECIAIS (Otimização)
    // ════════════════════════════════════════════════════════════
    lastCheckedDate : DATE := DATE#1970-01-01;      // Última data verificada
    cachedSpecialDateLimit : REAL := -1.0;          // -1 = inválido

    // ════════════════════════════════════════════════════════════
    // AUXILIARES
    // ════════════════════════════════════════════════════════════
    i : UINT;
END_VAR

    // ════════════════════════════════════════════════════════════════
    // 1. LEITURA DO RELÓGIO DO SISTEMA (UTC)
    // ════════════════════════════════════════════════════════════════

    GVL_Main.timestampUTC := TO_UDINT(SysTimeRtcGet(GVL_Main.Result));

    GVL_ALARM_MANAGER.CRIT_RTC_FAIL:=(GVL_Main.Result <> eResultCode.OK);
    IF GVL_ALARM_MANAGER.CRIT_RTC_FAIL THEN
        // ❌ ERRO: Relógio não disponível
        GVL_Main.MaxExportLimit := 0.0;
    	FC_LogEvent(
    		eCode:=E_EventCode.CRIT_RTC_FAILED,
    		bRaised:=TRUE,
    		rParam1:=0.0,
    		rParam2:=0.0,
    		uMachState := GVL_Main.MachineState
    		);
        RETURN;
    END_IF

    // ════════════════════════════════════════════════════════════════
    // 2. CÁLCULO DO OFFSET TOTAL (Fuso + Horário de Verão)
    // ════════════════════════════════════════════════════════════════

    // Offset base (fuso horário em segundos)
    offsetSeconds := GVL_Main.TIMEZONEOFFSET * 3600;  // Ex: -3 * 3600 = -10800

    // Adiciona horário de verão se ativo
    IF GVL_Persis.bHorarioVerao THEN
        offsetSeconds := offsetSeconds + 3600;      // +1 hora
    END_IF

    // ════════════════════════════════════════════════════════════════
    // 3. APLICA OFFSET AO TIMESTAMP UTC
    // ════════════════════════════════════════════════════════════════

    // ✅ MÉTODO SEGURO: Usa valor absoluto e subtrai/soma conforme sinal
    offsetSeconds_ABS := DINT_TO_UDINT(ABS(offsetSeconds));

    IF offsetSeconds < 0 THEN
        // Fuso NEGATIVO (Américas): subtrai
        timestampLocal_UDINT := GVL_Main.timestampUTC - offsetSeconds_ABS;
    ELSE
        // Fuso POSITIVO (Europa, Ásia): soma
        timestampLocal_UDINT := GVL_Main.timestampUTC + offsetSeconds_ABS;
    END_IF

    // ════════════════════════════════════════════════════════════════
    // 4. CONVERTE TIMESTAMP PARA DATA/HORA LOCAL
    // ════════════════════════════════════════════════════════════════

    dtNowLocal := UDINT_TO_DT(timestampLocal_UDINT);
    dataNowLocal := TO_DATE(dtNowLocal);

    // Extrai hora (0..23)
    todNowLocal := DT_TO_TOD(dtNowLocal);
    todAsDword := TOD_TO_DWORD(todNowLocal);
    hora := DWORD_TO_INT(todAsDword / DWORD#3600000);

    // Extrai dia da semana (1=Dom .. 7=Sáb)
    diadasemana := UDINT_TO_INT(((timestampLocal_UDINT / 86400) + 4) MOD 7) + 1;

    // ════════════════════════════���═══════════════════════════════════
    // 5. VERIFICA MUDANÇA DE DATA (Para atualizar cache)
    // ════════════════════════════════════════════════════════════════

    IF dataNowLocal <> lastCheckedDate THEN

        lastCheckedDate := dataNowLocal;
        cachedSpecialDateLimit := -1.0;  // Invalida cache

        FOR i := 1 TO GVL_Main.NDATASESPECIAIS DO

            // ✅ OTIMIZAÇÃO: Early exit se encontrar data vazia
            IF GVL_Persis.DatasEspeciais[i] = DATE#1970-01-01 THEN
                EXIT;  // Resto do array está vazio
            END_IF

            // Verifica se é data especial
            IF GVL_Persis.DatasEspeciais[i] = dataNowLocal THEN
                cachedSpecialDateLimit := GVL_Persis.SpecialDaySchedule[i];
                EXIT;  // Encontrou, pára a busca
            END_IF

        END_FOR

    END_IF

    // ════════════════════════════════════════════════════════════════
    // 6. USA CACHE DE DATA ESPECIAL (Se válido)
    // ════════════════════════════════════════════════════════════════

    IF cachedSpecialDateLimit >= 0.0 THEN
        // Data especial ativa
        GVL_Main.MaxExportLimit := cachedSpecialDateLimit;
    	FC_LogEvent(
    		eCode:=E_EventCode.INFO_SPECIAL_DATE_ACTIVE,
    		bRaised:=TRUE,
    		rParam1:=0.0,
    		rParam2:=0.0,
    		uMachState := GVL_Main.MachineState
    		);
        RETURN;																				// se é data especial, não olha busca por dia e hora, aborta
    END_IF

    // ════════════════════════════════════════════════════════════════
    // 7. AGENDA SEMANAL (Hora Local)
    // ════════════════════════════════════════════════════════════════

    // ✅ VALIDAÇÃO: Verifica se índices estão dentro dos limites
    semanaindex:= (diadasemana >= 1 AND diadasemana <= 7) AND (hora >= 0 AND hora <= 23);
    GVL_ALARM_MANAGER.CRIT_SCHEDULE_INDEX_INVALID:= NOT semanaindex;

    IF semanaindex THEN
        GVL_Main.MaxExportLimit := GVL_Persis.WeekSchedule_kW[diadasemana, hora + 1];     // Acessa agenda semanal
    ELSE																				  // ❌ ERRO: Índice inválido (não deveria ocorrer)
        GVL_Main.MaxExportLimit := 0.0;
    	FC_LogEvent(
    		eCode:=E_EventCode.CRIT_SCHEDULE_INDEX_INVALID,
    		bRaised:=TRUE,
    		rParam1:=0.0,
    		rParam2:=0.0,
    		uMachState := GVL_Main.MachineState
    		);

    END_IF
END_FUNCTION_BLOCK
